// TIA Portal project "speed_control_V2.5_e_V15" (V15)

(* hardware
DEVICE "GSD device_1"  GSD.Device.PN
   slot 0: "Rack"  Rail  V1.0
   slot 0: "s712xxsewgateway"  Gateway DFE32B V1.2  182x xxx x  V1.2
      slot 0: "Gateway DFE32B V1.2"  182x xxx x  V1.2
DEVICE "SIMATIC 1200 station_2"  S71200.Device
   slot 0: "S7-1200 rack"  Rack  V1.0
   slot 1: "s712xx"  CPU 1211C AC/DC/Rly  6ES7 211-1BD30-0XB0  V2.0
*)

// ===== PLC "s712xx"  CPU 1211C AC/DC/Rly =====

DATA_BLOCK "Drive_2_272"   // DB272
{ S7_Optimized_Access := 'FALSE' }
VERSION : 0.1
   VAR
      IO_ADDRESS_or_HW_IDENTIFIER : Int := 291;   // S73xx/4xx: Assign Peripheral Address; S7 1x00: assign HW_Identifier
      ENABLE_RAPID_STOP : Bool;
      ENABLE : Bool;
      RESET : Bool;
      SETPOINT_SPEED : Int;
      RAMP : Int := 10000;   // Attention: Avoid ramp =0!
      COMMUNICATION_OK : Bool;
      INVERTER_READY : Bool;
      FAULT_OF_AXIS : Bool;
      FAULT_NO : Int;
      ACTUAL_SPEED : Int;
      OUTPUT_CURRENT : Int;
   END_VAR
BEGIN
END_DATA_BLOCK

DATA_BLOCK "Drive_1_281"   // DB281
{ S7_Optimized_Access := 'FALSE' }
VERSION : 0.1
   VAR
      IO_ADDRESS_or_HW_IDENTIFIER : Int := 281;   // S73xx/4xx: Assign Peripheral Address; S7 1x00: assign HW_Identifier
      ENABLE_RAPID_STOP : Bool;
      ENABLE : Bool;
      RESET : Bool;
      SETPOINT_SPEED : Int;
      RAMP : Int := 10000;   // Attention: Avoid ramp =0!
      COMMUNICATION_OK : Bool;
      INVERTER_READY : Bool;
      FAULT_OF_AXIS : Bool;
      FAULT_NO : Int;
      ACTUAL_SPEED : Int;
      OUTPUT_CURRENT : Int;
   END_VAR
BEGIN
END_DATA_BLOCK

FUNCTION "Call_speed_control" : Void   // FC100, FBD
TITLE = Call "speed_control_S71xxx" & "speed_control_S71xxx_scl"
{ S7_Optimized_Access := 'FALSE' }
VERSION : 0.1
// This sample program shows the basic approach only.
// We do not accept legal or other liability for
// incorrect program functions and their consequences!
// 
// For project planning and startup of the MC07 series on PROFIBUS DP and PROFINET 
// IO, see the following documentation:
// - MC07 system manual
// - Manual Fieldbus Interface DFP21B and DFE32B
// - MC07 communication manual
// 
// In the hardware configuration, eight drives were configured with the module 
// "One Module per drive." Each of the eight drives has been assigned a slot and a 
// discrete periphery area. We are calling up the first drive in this function as 
// an example
BEGIN

REGION Network 1: Controll drive 1, call FC133 "speed_control_S71xxx"
   // This function FC133 "speed_control_S71xxx" can be used to control the MOVITRAC frequency inverters on 
   // PROFIBUS DP in conjunction with the Gateway DFP21B or PROFINET IO in 
   // confunction with the gateway DFE32B.
   // 
   // The following parameters deviate from the factory setting:
   // P100/101 Setpoint source/control source => SBUS;
   // P881 SBUS address <> 0; see manual "Fieldbus Interface DFP21B"
   // P872 Setpoint description PO3 => Ramp
   // => P876 Enable PO data = ON
   // "Drive_IO_Address": Start address of the I/O area => hardware configuration
   // 
   // FC inputs:
   // Attention: "HW_IDENTIFIER"   S7 1x00: Hardware Identifier  of the correspondening slot;
   // Enable of drive:
   // Enable via dig. inputs (CW/Stop & Enable/Stop) & 
   // Enable via control word (Enable_rapid_stop & Enable)
   // "Reset" = true: Confirm error
   // "SETPOINT_SPEED": Preset of set speed in rpm (integer),
   // "RAMP": Preset of ramp in ms (integer)
   // 
   // FC outputs:
   // If data transmission/PROFIBUS is faulty, all outputs will be deleted.
   // => "Communication_OK" = false (self-confirming)
   // "INVERTER_READY" = true: No error present & mains voltage ON
   // "FAULT_OF_AXIS" = true: Error is present.
   // "FAULT_NO" <> 0: The error codes are listed in the system manual and are 
   // displayed 
   // in MOVITOOLS (status, bus monitor).
   // "ACTUAL_SPEED": Actual speed (INT) in rpm
   // "OUTPUT_CURRENT": Apparent current (INT) in percentage of rated unit current
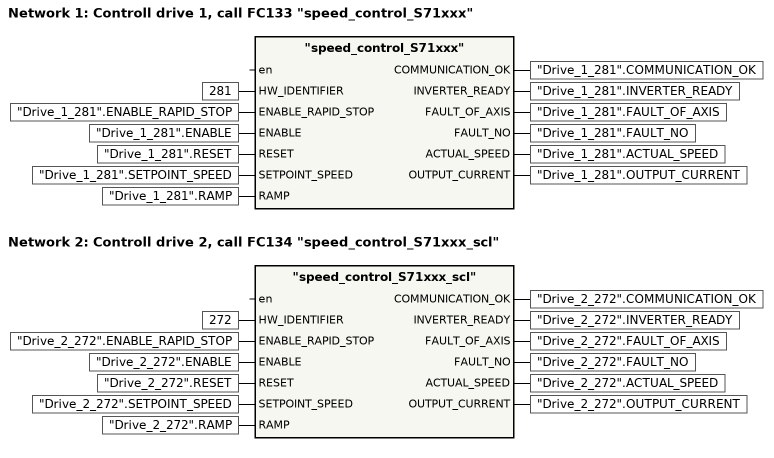
   "speed_control_S71xxx"(HW_IDENTIFIER := 281,
                          ENABLE_RAPID_STOP := "Drive_1_281".ENABLE_RAPID_STOP,
                          ENABLE := "Drive_1_281".ENABLE,
                          RESET := "Drive_1_281".RESET,
                          SETPOINT_SPEED := "Drive_1_281".SETPOINT_SPEED,
                          RAMP := "Drive_1_281".RAMP,
                          COMMUNICATION_OK => "Drive_1_281".COMMUNICATION_OK,
                          INVERTER_READY => "Drive_1_281".INVERTER_READY,
                          FAULT_OF_AXIS => "Drive_1_281".FAULT_OF_AXIS,
                          FAULT_NO => "Drive_1_281".FAULT_NO,
                          ACTUAL_SPEED => "Drive_1_281".ACTUAL_SPEED,
                          OUTPUT_CURRENT => "Drive_1_281".OUTPUT_CURRENT);
END_REGION

REGION Network 2: Controll drive 2, call FC134 "speed_control_S71xxx_scl"
   // This function FC134 "speed_control_S71xxx_scl" can be used to control the MOVITRAC frequency inverters on 
   // PROFIBUS DP in conjunction with the Gateway DFP21B or PROFINET IO in 
   // confunction with the gateway DFE32B.
   // 
   // The following parameters deviate from the factory setting:
   // P100/101 Setpoint source/control source => SBUS;
   // P881 SBUS address <> 0; see manual "Fieldbus Interface DFP21B"
   // P872 Setpoint description PO3 => Ramp
   // => P876 Enable PO data = ON
   // 
   // FC inputs:
   // "HW_IDENTIFIER"   S7 1x00: Assign Hardware Identifier of the correspondening slot;
   // Enable of drive:
   // Enable via dig. inputs (CW/Stop & Enable/Stop) & 
   // Enable via control word (Enable_rapid_stop & Enable)
   // "Reset" = true: Confirm error
   // "SETPOINT_SPEED": Preset of set speed in rpm (integer),
   // "RAMP": Preset of ramp in ms (integer)
   // 
   // FC outputs:
   // If data transmission/PROFIBUS is faulty, all outputs will be deleted.
   // => "Communication_OK" = false (self-confirming)
   // "INVERTER_READY" = true: No error present & mains voltage ON
   // "FAULT_OF_AXIS" = true: Error is present.
   // "FAULT_NO" <> 0: The error codes are listed in the system manual and are 
   // displayed 
   // in MOVITOOLS (status, bus monitor).
   // "ACTUAL_SPEED": Actual speed (INT) in rpm
   // "OUTPUT_CURRENT": Apparent current (INT) in percentage of rated unit current
   "speed_control_S71xxx_scl"(HW_IDENTIFIER := 272,
                           ENABLE_RAPID_STOP := "Drive_2_272".ENABLE_RAPID_STOP,
                           ENABLE := "Drive_2_272".ENABLE,
                           RESET := "Drive_2_272".RESET,
                           SETPOINT_SPEED := "Drive_2_272".SETPOINT_SPEED,
                           RAMP := "Drive_2_272".RAMP,
                           COMMUNICATION_OK => "Drive_2_272".COMMUNICATION_OK,
                           INVERTER_READY => "Drive_2_272".INVERTER_READY,
                           FAULT_OF_AXIS => "Drive_2_272".FAULT_OF_AXIS,
                           FAULT_NO => "Drive_2_272".FAULT_NO,
                           ACTUAL_SPEED => "Drive_2_272".ACTUAL_SPEED,
                           OUTPUT_CURRENT => "Drive_2_272".OUTPUT_CURRENT);
END_REGION
END_FUNCTION

FUNCTION "speed_control_S71xxx" : Void   // FC133, FBD
TITLE = speed_control
{ S7_Optimized_Access := 'FALSE' }
AUTHOR : SE-PAS
FAMILY : PROFIBUS
NAME : MC07
VERSION : 2.4
// This sample program shows the basic approach only.
// We do not accept legal or other liability for
// incorrect program functions and their consequences!
// 
// 
// This function FC133 "speed_control_S71xxx"can be used to control the MOVITRAC frequency inverters on PROFIBUS DP in conjunction with the Gateway DFP21B or PROFINET IO in 
// confunction with the gateway DFE32B.
// 
// The following parameters deviate from the factory setting:
// P100/101 Setpoint source/control source => SBUS;
// P881 SBUS address <> 0; see manual "Fieldbus Interface DFP21B"
// P872 Setpoint description PO3 => Ramp
// => P876 Enable PO data = ON
// 
// FC inputs:
// "HW_IDENTIFIER"   S7 1x00: assign HW_Identifier of the correspondending slot
// Enable of drive:
// Enable via dig. inputs (CW/Stop & Enable/Stop) & 
// Enable via control word (Enable_rapid_stop & Enable)
// "Reset" = true: Confirm error
// "SETPOINT_SPEED": Preset of set speed in rpm (integer),
// "RAMP": Preset of ramp in ms (integer)
// 
// FC outputs:
// If data transmission/PROFIBUS is faulty, all outputs will be deleted.
// => "Communication_OK" = false (self-confirming)
// "INVERTER_READY" = true: No error present & mains voltage ON
// "FAULT_OF_AXIS" = true: Error is present.
// "FAULT_NO" <> 0: The error codes are listed in the system manual and are 
// displayed 
// in MOVITOOLS (status, bus monitor).
// "ACTUAL_SPEED": Actual speed (INT) in rpm
// "OUTPUT_CURRENT": Apparent current (INT) in percentage of rated unit current
// Dieses Programmbeispiel zeigt nur die prinzipielle Vorgehensweise.
// Für fehlerhafte Programmfunktionen und deren Folgen
// kann weder eine juristische, noch irgendeine Haftung übernommen werden!
// 
// Diese Funktion kann für PROFIBUS DP oder PROFINET I/O genutzt werden
   VAR_INPUT
      HW_IDENTIFIER : Hw_Io;   // S7 1x00: assign HW_Identifier
      ENABLE_RAPID_STOP : Bool;
      ENABLE : Bool;
      RESET : Bool;
      SETPOINT_SPEED : Int;
      RAMP : Int;
   END_VAR
   VAR_OUTPUT
      COMMUNICATION_OK : Bool;   // SFC14/SFC15: Return Value = 0
      INVERTER_READY : Bool;
      FAULT_OF_AXIS : Bool;
      FAULT_NO : Int;
      ACTUAL_SPEED : Int;
      OUTPUT_CURRENT : Int;
   END_VAR
   VAR_TEMP
      PI : Struct
         STATUS : Byte;
         ENABLE_OUTPUT_STAGE : Bool;
         INVERTER_READY : Bool;
         PO_DATA_ENABLE : Bool;
         STW_Bit_3 : Bool;
         STW_Bit_4 : Bool;
         ERROR : Bool;
         STW_Bit_6 : Bool;
         STW_Bit_7 : Bool;
         ACTUAL_SPEED : Int;
         OUTPUT_CURRENT : Int;
      END_STRUCT;
      PO : Struct
         DIRECTION_MOTOR_POTI : Bool;
         MOTOR_POTI_UP : Bool;
         MOTOR_POTI_DOWN : Bool;
         FIXED_INTERNAL_SETPOINTS : Bool;
         FIXED_INTERNAL_SETP_1 : Bool;
         FIXED_SETP_SWITCHOVER : Bool;
         CTW_Bit_14 : Bool;
         CTW_Bit_15 : Bool;
         CONTR_INHIBIT : Bool;
         RAPID_STOP : Bool;
         STOP : Bool;
         CTW_Bit_3 : Bool;
         CTW_Bit_4 : Bool;
         CTW_Bit_5 : Bool;
         RESET_FAULT : Bool;
         CTW_Bit_7 : Bool;
         SETPOINT_SPEED : Int;
         RAMP : Int;
      END_STRUCT;
      RETURNCODE_SFC14 : Int;
      RETURNCODE_SFC15 : Int;
      Com_SFC14_OK : Bool;
      Com_SFC15_OK : Bool;
      FALSE : Bool;
   END_VAR
   VAR_TEMP   // added for the SCL form of the ladder/FBD networks
      _w1 : Bool;
   END_VAR
BEGIN

REGION Network 1: Def. "#FALSE"
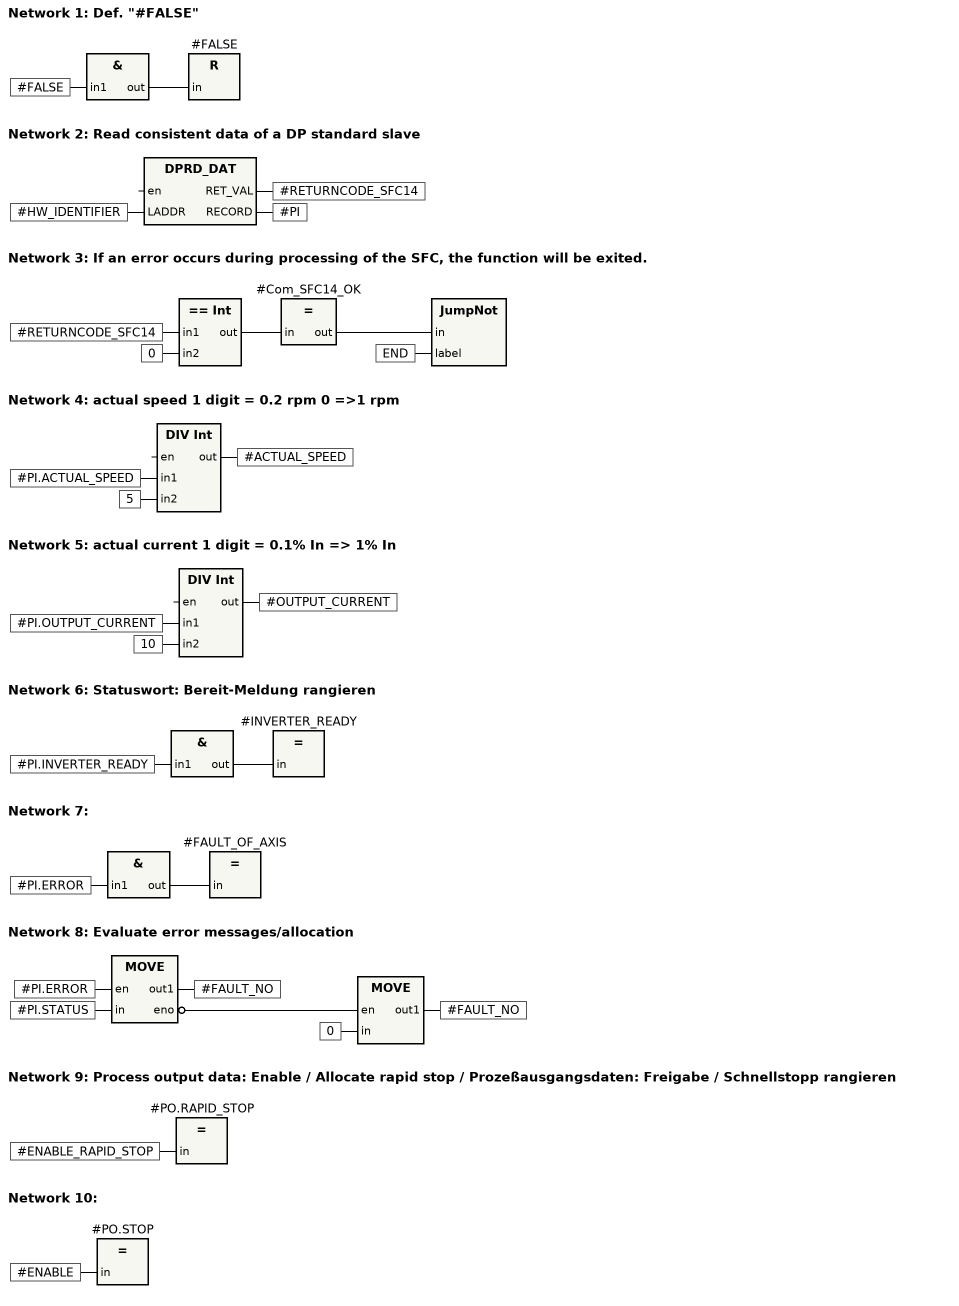
   IF #FALSE THEN #FALSE := FALSE; END_IF;
END_REGION

REGION Network 2: Read consistent data of a DP standard slave
   #RETURNCODE_SFC14 := DPRD_DAT(LADDR := #HW_IDENTIFIER, RECORD => #PI);
END_REGION

REGION Network 3: If an error occurs during processing of the SFC, the function will be exited.
   // no SCL statement known for JumpNot: written as a call
   #Com_SFC14_OK := #RETURNCODE_SFC14 = 0;
   JumpNot(in := #Com_SFC14_OK, label := END);
END_REGION

REGION Network 4: actual speed 1 digit = 0.2 rpm 0 =>1 rpm
   #ACTUAL_SPEED := #PI.ACTUAL_SPEED / 5;
END_REGION

REGION Network 5: actual current 1 digit = 0.1% In => 1% In
   #OUTPUT_CURRENT := #PI.OUTPUT_CURRENT / 10;
END_REGION

REGION Network 6: Statuswort: Bereit-Meldung rangieren
   #INVERTER_READY := #PI.INVERTER_READY;
END_REGION

REGION Network 7
   #FAULT_OF_AXIS := #PI.ERROR;
END_REGION

REGION Network 8: Evaluate error messages/allocation
   // If an error bit has been set, an error number will be issued.
   // If no error is present, a zero will be issued.
   // ENO of a box is taken as its EN; it also drops when the box reports an error
   IF #PI.ERROR THEN #FAULT_NO := #PI.STATUS; END_IF;
   IF NOT #PI.ERROR THEN #FAULT_NO := 0; END_IF;
END_REGION

REGION Network 9: Process output data: Enable / Allocate rapid stop / Prozeßausgangsdaten: Freigabe / Schnellstopp rangieren
   #PO.RAPID_STOP := #ENABLE_RAPID_STOP;
END_REGION

REGION Network 10
   #PO.STOP := #ENABLE;
END_REGION

REGION Network 11: Fault_Reset
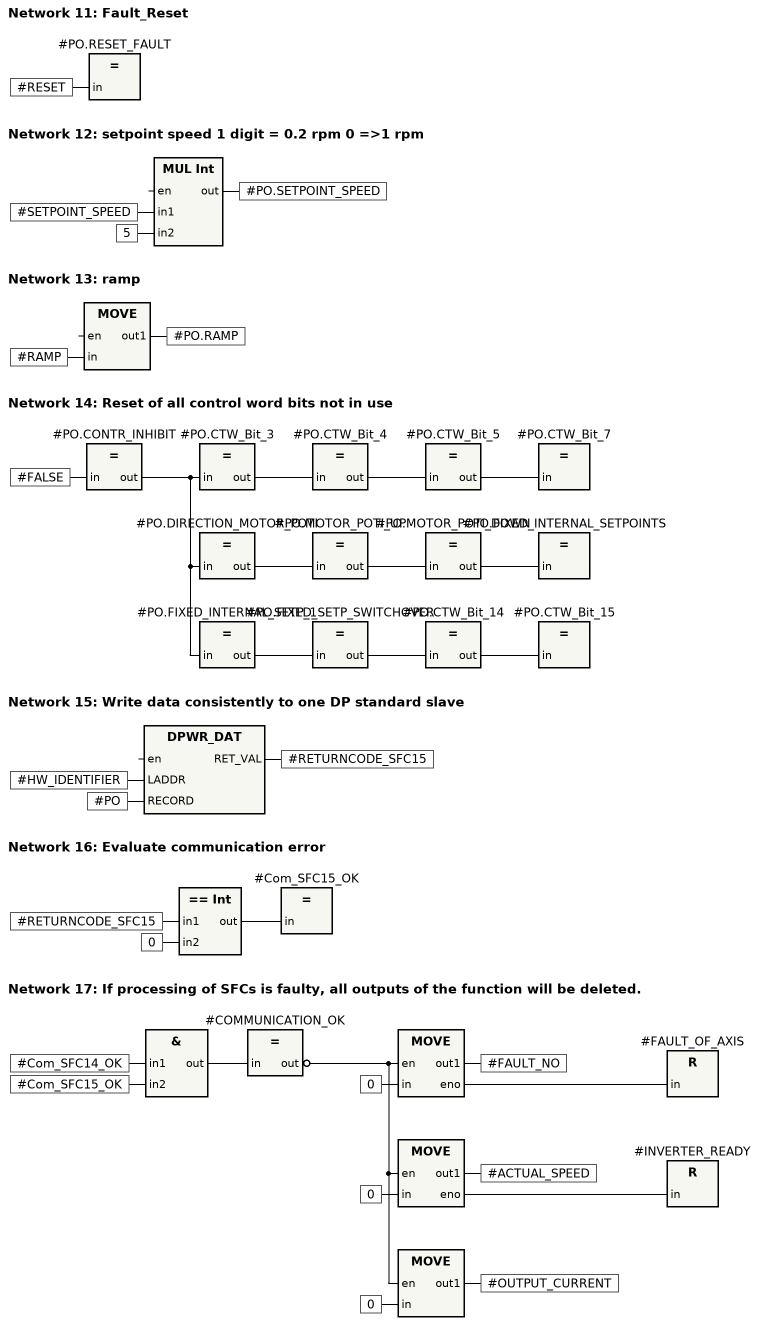
   #PO.RESET_FAULT := #RESET;
END_REGION

REGION Network 12: setpoint speed 1 digit = 0.2 rpm 0 =>1 rpm
   #PO.SETPOINT_SPEED := #SETPOINT_SPEED * 5;
END_REGION

REGION Network 13: ramp
   #PO.RAMP := #RAMP;
END_REGION

REGION Network 14: Reset of all control word bits not in use
   #PO.CONTR_INHIBIT := #FALSE;
   #PO.CTW_Bit_3 := #FALSE;
   #PO.CTW_Bit_4 := #FALSE;
   #PO.CTW_Bit_5 := #FALSE;
   #PO.CTW_Bit_7 := #FALSE;
   #PO.DIRECTION_MOTOR_POTI := #FALSE;
   #PO.MOTOR_POTI_UP := #FALSE;
   #PO.MOTOR_POTI_DOWN := #FALSE;
   #PO.FIXED_INTERNAL_SETPOINTS := #FALSE;
   #PO.FIXED_INTERNAL_SETP_1 := #FALSE;
   #PO.FIXED_SETP_SWITCHOVER := #FALSE;
   #PO.CTW_Bit_14 := #FALSE;
   #PO.CTW_Bit_15 := #FALSE;
END_REGION

REGION Network 15: Write data consistently to one DP standard slave
   #RETURNCODE_SFC15 := DPWR_DAT(LADDR := #HW_IDENTIFIER, RECORD := #PO);
END_REGION

REGION Network 16: Evaluate communication error
   #Com_SFC15_OK := #RETURNCODE_SFC15 = 0;
END_REGION

REGION Network 17: If processing of SFCs is faulty, all outputs of the function will be deleted.
   // ENO of a box is taken as its EN; it also drops when the box reports an error
   END:
   #_w1 := #Com_SFC14_OK AND #Com_SFC15_OK;
   #COMMUNICATION_OK := #_w1;
   IF NOT #_w1 THEN
       #FAULT_NO := 0;
       #FAULT_OF_AXIS := FALSE;
       #ACTUAL_SPEED := 0;
       #INVERTER_READY := FALSE;
       #OUTPUT_CURRENT := 0;
   END_IF;
END_REGION
END_FUNCTION

FUNCTION "speed_control_S71xxx_scl" : Void   // FC134, SCL
{ S7_Optimized_Access := 'FALSE' }
VERSION : 0.1
   VAR_INPUT
      HW_IDENTIFIER : Hw_Io;   // S7 1x00: assign HW_Identifier
      ENABLE_RAPID_STOP : Bool;
      ENABLE : Bool;
      RESET : Bool;
      SETPOINT_SPEED : Int;
      RAMP : Int;
   END_VAR
   VAR_OUTPUT
      COMMUNICATION_OK : Bool;   // SFC14/SFC15: Return Value = 0
      INVERTER_READY : Bool;
      FAULT_OF_AXIS : Bool;
      FAULT_NO : Int;
      ACTUAL_SPEED : Int;
      OUTPUT_CURRENT : Int;
   END_VAR
   VAR_TEMP
      PI : Struct
         STATUS : Byte;
         ENABLE_OUTPUT_STAGE : Bool;
         INVERTER_READY : Bool;
         PO_DATA_ENABLE : Bool;
         STW_Bit_3 : Bool;
         STW_Bit_4 : Bool;
         ERROR : Bool;
         STW_Bit_6 : Bool;
         STW_Bit_7 : Bool;
         ACTUAL_SPEED : Int;
         OUTPUT_CURRENT : Int;
      END_STRUCT;
      PO : Struct
         DIRECTION_MOTOR_POTI : Bool;
         MOTOR_POTI_UP : Bool;
         MOTOR_POTI_DOWN : Bool;
         FIXED_INTERNAL_SETPOINTS : Bool;
         FIXED_INTERNAL_SETP_1 : Bool;
         FIXED_SETP_SWITCHOVER : Bool;
         CTW_Bit_14 : Bool;
         CTW_Bit_15 : Bool;
         CONTR_INHIBIT : Bool;
         RAPID_STOP : Bool;
         STOP : Bool;
         CTW_Bit_3 : Bool;
         CTW_Bit_4 : Bool;
         CTW_Bit_5 : Bool;
         RESET_FAULT : Bool;
         CTW_Bit_7 : Bool;
         SETPOINT_SPEED : Int;
         RAMP : Int;
      END_STRUCT;
      DPRD_RET_VAL : Int;   // Return Value DPRD_DAT; <> 0 => error
      DPWR_RET_VAL : Int;   // Return Valoe: DPWR_DAT; <> 0 => error
      Com_SFC14_OK : Bool;
      Com_SFC15_OK : Bool;
   END_VAR
BEGIN
   //This sample program shows the basic approach only.
   //We do not accept legal or other liability for
   //incorrect program functions and their consequences!
   //
   (*This function FC134 "speed_control_S71xxx_scl" can be used to control the MOVITRAC frequency inverters on 
   PROFIBUS DP in conjunction with the Gateway DFP21B or PROFINET IO in 
   confunction with the gateway DFE32B.

   The following parameters deviate from the factory setting:
   P100/101 Setpoint source/control source => SBUS;
   P881 SBUS address <> 0; see manual "Fieldbus Interface DFP21B"
   P872 Setpoint description PO3 => Ramp
   => P876 Enable PO data = ON

   FC inputs:
   "HW_IDENTIFIER"   S7 1x00: Assign Hardware Identifier of the correspondening slot;
   Enable of drive:
   Enable via dig. inputs (CW/Stop & Enable/Stop) & 
   Enable via control word (Enable_rapid_stop & Enable)
   "Reset" = true: Confirm error
   "SETPOINT_SPEED": Preset of set speed in rpm (integer),
   "RAMP": Preset of ramp in ms (integer)

   FC outputs:
   If data transmission/PROFIBUS is faulty, all outputs will be deleted.
   => "Communication_OK" = false (self-confirming)
   "INVERTER_READY" = true: No error present & mains voltage ON
   "FAULT_OF_AXIS" = true: Error is present.
   "FAULT_NO" <> 0: The error codes are listed in the system manual and are 
   displayed 
   in MOVITOOLS (status, bus monitor).
   "ACTUAL_SPEED": Actual speed (INT) in rpm
   "OUTPUT_CURRENT": Apparent current (INT) in percentage of rated unit current*)

   #DPRD_RET_VAL := DPRD_DAT(LADDR := #HW_IDENTIFIER, RECORD => #PI);//DPRD_DAT: Read consistent data

   IF #DPRD_RET_VAL = 0 THEN
       #COMMUNICATION_OK := true;//IF no error occurs WHILE the instruction DPRD_DAT is being executed THEN...

       #ACTUAL_SPEED := #PI.ACTUAL_SPEED/5; //actual speed 1 digit = 0.2 rpm  
       #OUTPUT_CURRENT := #PI.OUTPUT_CURRENT/10;//actual current 1 digit = 0.1% In => 1% In

       #INVERTER_READY := #PI.INVERTER_READY;
       #FAULT_OF_AXIS := #PI.ERROR;

       IF #PI.ERROR = true THEN
           #FAULT_NO := #PI.STATUS;
       ELSE
           #FAULT_NO := 0;
       END_IF; //depending on the error-bit =1 the fault_no is displayed; else fault = 0; 
       //Control bits:
       #PO.RAPID_STOP := #ENABLE_RAPID_STOP;
       #PO.STOP := #ENABLE;
       #PO.RESET_FAULT := #RESET;
       //convert and assign "analog"-values:
       #PO.SETPOINT_SPEED := #SETPOINT_SPEED * 5;//actual speed 1 digit = 0.2 rpm  
       #PO.RAMP := #RAMP;

       //Reset of all control word bits not in use:
       #PO.CONTR_INHIBIT := false;
       #PO.CTW_Bit_3 := false;
       #PO.CTW_Bit_4 := false;
       #PO.CTW_Bit_5 := false;
       #PO.CTW_Bit_7 := false;
       #PO.DIRECTION_MOTOR_POTI := false;
       #PO.MOTOR_POTI_UP := false;
       #PO.MOTOR_POTI_DOWN:=false;
       #PO.FIXED_INTERNAL_SETPOINTS := false;
       #PO.FIXED_INTERNAL_SETP_1:=false;
       #PO.FIXED_SETP_SWITCHOVER := false;
       #PO.CTW_Bit_14 := false;
       #PO.CTW_Bit_15 := false;
   ELSE
       GOTO END; //If an error occurs during processing of the DP_RD_DAT-function, the function will be exited

   END_IF;

   #DPWR_RET_VAL := DPWR_DAT(LADDR := #HW_IDENTIFIER, RECORD := #PO);//DPWR_DAT: Write consistent data of a DP standard slave 

   END:
   IF #DPRD_RET_VAL <> 0 OR #DPWR_RET_VAL <> 0 THEN
       #COMMUNICATION_OK := false; //all outputs will be deleted, if processing of the DPRD_DAT or DPWR_DA-function is faulty
       #INVERTER_READY := false;
       #FAULT_OF_AXIS := false;
       #FAULT_NO := 0;
       #ACTUAL_SPEED := 0;
       #OUTPUT_CURRENT := 0; 
   END_IF;
END_FUNCTION

ORGANIZATION_BLOCK "Main"   // OB1, FBD, ProgramCycle
TITLE = "Main Program Sweep (Cycle)"
{ S7_Optimized_Access := 'TRUE' }
VERSION : 0.1
// This TIA- project demonstrates how to incorporate the MOVITRAC inverter series in the SIMATIC TIA-world.
// A function FC130 can be used to control the MOVITRAC frequency inverters on PROFINET IO in 
// conjunction with the Gateway DFE32B or PROFIBUS DP in conjunction with the Gateway DFP21B:
// 
// The sample blocks do not have "optimized block access" so that they can be used downwards compatible with the S73xx and S74xx CPUs.
// An S712xx controller and an S73xx controller are integrated in the PROFINET network.
// One DFE gateway is assigned to each PROFINET controller:
//                               
//                               device number 1         device number 2
//                               
//            CPU 12xx           DFE32B-Gateway         DFE32B-Gateway        CPU3xx
//                            (assigned "12xx")     (assigned "3xx")              
// PROFINET-           
// device name:"12xx"         "s712xxsewgateway"       "s73xxsewgateway"      "3xx"
//                I_____________________I_____________________I_________________I
//                                Ethernet                          Ethernet                       Ethernet
BEGIN

REGION Network 1
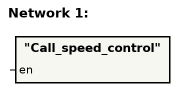
   "Call_speed_control"();
END_REGION
END_ORGANIZATION_BLOCK